TYPE ST_AXIS_POSITION :
STRUCT
END_STRUCT
END_TYPE

(* stored: Version 1.1.0.1, ProductVersion 3.1.4024.11
   DUT ST_AXIS_POSITION: Id {6d45ea76-2343-44a1-9ef7-6b223a81beb3} *)
